// TIA Portal V20 export
// export: Created 2025-12-01T14:57:45.4290104Z, ExportSetting None, DisplayName Totally Integrated Automation Portal, DisplayVersion V20 Update 3, DisplayName TIA Portal Openness, DisplayVersion V20 Update 3, DisplayName TIA Portal Version Control Interface, DisplayVersion V20 Update 3, DisplayName STEP 7 Professional, DisplayVersion V20 Update 3, DisplayName STEP 7 Safety, DisplayVersion V20 Update 2, DisplayName WinCC Basic/Comfort/Advanced, DisplayVersion V20 Update 3, DisplayName WinCC Professional, DisplayVersion V20 Update 3, DisplayName WinCC Unified, DisplayVersion V20 Update 3
FUNCTION "FC824_Recoge_Eventos_Routing" : Void   // FC824, LAD
TITLE = recoge eventos router
{ S7_Optimized_Access := 'FALSE' }
AUTHOR : NRF
FAMILY : Routing
VERSION : 1.0
// recoge del DB de recepción de mensajes todos los mensajes dirigidos al sistema routing y los extrae y escribe en un DB independiente para su posterior tratamiento
// stored: AutoNumber false, SetENOAutomatically false
   VAR_INPUT
      NumJdT : UInt;
      DBEventosrouter : Word;
   END_VAR
   VAR_IN_OUT
      PunteroEventos : DWord;   // Puntero al DB de Eventos Recibidos
   END_VAR
   VAR_TEMP
      DBEventosRec : Word;   // DB de Eventos Recibidos
      Numero_bytes : UInt;
      retval : Int;
      inicio_destino : Int;
      inicio_origen : Int;
      origen : Any;
      destino : Any;
      Contador : Int;
   END_VAR
BEGIN

NETWORK
TITLE = Inicializar
/////////////////////////////////////////////////////////////////////////
/// --- Comprobar que JDT

      SET;
      L     "JDT1_NDB_EventosRec";  // Cogemos el DB de Eventos Recibidos
      T     #DBEventosRec;

/////////////////////////////////////////////////////////////////////////

      L     #NumJdT;
      L     2;
      <>I;
      JC    NoJdT02;

/////////////////////////////////////////////////////////////////////////

      SET;
      L     "JDT2_NDB_EventosRec";  // Cogemos el DB de Eventos Recibidos
      T     #DBEventosRec;

NoJdT02:NOP   0;

/////////////////////////////////////////////////////////////////////////



NETWORK
TITLE = Distribucion de los Eventos (LIsta del DB de Conversion)
/////////////////////////////////////////////////////////////////////////
/////////////////////////////////////////////////////////////////////////
/////////////////////////////////////////////////////////////////////////
// Hay que recoger el Evento, para despues repartir
// Despues '{' va el tipo de eventos (2 Bytes)
      L     #PunteroEventos;  // Recogo por donde va empieza el evento
      LAR2;  // del Router


// el objetivo es recoger todo el evento y volcarlo en un DB independiente
// del que luego el router hará el tratamiento
// inicializamos el contador a 0 y vamos contando cuantos bytes copiar

      L     0;
      T     #Numero_bytes;

      OPN   DB [#DBEventosRec];

bucle:NOP   0;
      A(;
      L     DBB [AR2, P#0.0];
      L     '}';
      ==I;
      );
      O(;
      L     DBB [AR2, P#0.0];
      L     0;
      ==I;
      );
      JC    copia;

      +AR2  P#1.0;


      L     #Numero_bytes;
      L     1;
      +I;
      T     #Numero_bytes;
      JU    bucle;

copia:NOP   0;

REGION Network 3 (SCL)
   // buscamos dentro del DB de eventos del router la primera posición libre para guardar el mensaje
   // 
   FOR #Contador := 1 TO 2500 DO
       IF "DB210_DB_Eventos_Router".EVENTO[#Contador] = ' ' THEN
           #inicio_destino := #Contador-1;
           IF #Contador > 1 THEN
               "DB210_DB_Eventos_Router".EVENTO[#Contador] := ';';
               #inicio_destino += 1;
           ELSE
               EXIT;
           END_IF;
           EXIT;
       ELSE IF #Contador= 2500 THEN
               RETURN;
           END_IF ;
       END_IF;
       END_FOR;
END_REGION

NETWORK
TITLE = realizar la copia en un DB independiente
////////////////////////////////////////////////////////
// iniciamos el proceso de copia



// generamos puntero de origen
// calculo la posicion incial

      L     #PunteroEventos;
      SRD   3;
      T     #inicio_origen;

      LAR1  P##origen;

      L     B#16#10;  // CARGAR EL ID DE SINTAXIS
      T     LB [AR1, P#0.0];

      L     B#16#2;  // CARGAR EL TIPO DE DATOS, POR DEFECTO BYTES
      T     LB [AR1, P#1.0];

      L     #Numero_bytes;  // CARGAR LA CANTIDAD DE BYTES A COPIAR
      T     LW [AR1, P#2.0];

      L     #DBEventosRec;
      T     LW [AR1, P#4.0];
// CARGO EL BYTE DETRABAJO
      L     #inicio_origen;  //CON ESTO LE INDICO A PARTIR DE QUE BYTE QUIERO QUE BORRE
      SLW   3;
      T     LD [AR1, P#6.0];
// LE INDICO QUE ES UN DB
      L     B#16#84;
      T     LB [AR1, P#6.0];

//=============================================================================
// genero el puntero al destino

      LAR1  P##destino;

      L     B#16#10;  // CARGAR EL ID DE SINTAXIS
      T     LB [AR1, P#0.0];

      L     B#16#2;  // CARGAR EL TIPO DE DATOS, POR DEFECTO BYTES
      T     LB [AR1, P#1.0];

      L     #Numero_bytes;  // CARGAR LA CANTIDAD DE BYTES A COPIAR
      T     LW [AR1, P#2.0];

      L     #DBEventosrouter;
      T     LW [AR1, P#4.0];
// CARGO EL BYTE DETRABAJO
      L     #inicio_destino;  //CON ESTO LE INDICO A PARTIR DE QUE BYTE QUIERO QUE BORRE
      SLW   3;
      T     LD [AR1, P#6.0];
// LE INDICO QUE ES UN DB
      L     B#16#84;
      T     LB [AR1, P#6.0];

//=============================================================================
      CALL  UBLKMOV
      ( SRCBLK  := #origen,
        RET_VAL := #retval,
        DSTBLK  := #destino
      );



      TAR2;  // Devuelve por donde va empieza el evento
      T     #PunteroEventos;  // del Router
      JU    FinalizarFuncion;

FinalizarFuncion:NOP   0;

END_FUNCTION
